// TwinCAT 3 PLC project GRAB
// ProgramVersion: 3.1.4024.12
// libraries:
//   CmpBitmapPool, * (System)
//   Tc2_MC2, * (Beckhoff Automation GmbH)
//   Tc2_Standard, * (Beckhoff Automation GmbH)
//   Tc2_System, * (Beckhoff Automation GmbH)
//   Tc3_Module, * (Beckhoff Automation GmbH)
//   VisuSymbols,3.5.10.0,System
// project tree:
//   / GlobalTextList.TcGTLO, ImagePool.TcIPO (not stored), PlcTask.TcTTO, Visualization Manager.TcVMO (not stored)
//   GVLs/ GVL.TcGVL, HAVL.TcGVL, RAVL.TcGVL, VAVL.TcGVL
//   POUs/ Homing.TcPOU, HorAxisPosCon.TcPOU, MAIN.TcPOU, ManualHorAxis.TcPOU, ManualRotAxis.TcPOU, ManualVerAxis.TcPOU, PositionHorAxis.TcPOU, PositionRotAxis.TcPOU, PositionVerAxis.TcPOU, POU.TcPOU, RunGRAB.TcPOU, Stop.TcPOU
//   VISUs/ Visualization.TcVIS
// real-time tasks:
//   TASK PlcTask: cycle T#10ms, priority 20, ADS port 350
// motion (NC):
//   TASK NC-Task 1 SAF: cycle T#2ms, priority 4, ADS port 501
//   TASK NC-Task 1 SVB: cycle T#10ms, priority 8, ADS port 511
//   AXIS HorizontalAxis (id 3)
//     Dynamic: AccelerationMaximum=2000, DecelerationMaximum=2000, Acceleration=100, Deceleration=500, Jerk=5000
//     Velo: RefSearch=80, RefSync=20, SlowManual=150, FastManual=150, Maximum=200
//     OtherSettings: AllowMotionCmdToSlave=true
//     encoder EncType=19
//       EncPara: ScaleFactorNumerator=0.004208, MaxCount=#xffffffff
//         SoftEndMinControl: Enable=true, Range=-100
//         SoftEndMaxControl: Enable=true, Range=700
//         Inc: RefSearchInverse=true, RefSyncInverse=false, RefSoftSyncMask=#x00000fff
//     drive DrvType=16
//       DrvPara: MaxCount=#xffffffff, DriveControlDWord=#x00020000
//         Analog: VeloReferenz=150, TorqueSetpointScale=10, ScaleFactorActTorque=0.1
//         TimeComp: TaskDelayCycles=1
//     controller CtrType=1
//       CtrPara: PriorControlFactor=1
//         PosDiffControl: Range=10
//         Observer: BandWidth=20
//   AXIS RotationAxis (id 4)
//     General: UnitName=Degree
//     Dynamic: AccelerationMaximum=20, DecelerationMaximum=20, Acceleration=10, Deceleration=50, Jerk=50
//     Velo: RefSearch=10, RefSync=5, SlowManual=20, FastManual=20, Maximum=21
//     OtherSettings: AllowMotionCmdToSlave=true, PulseDistancePos=0.05, PulseDistanceNeg=0.05
//     encoder EncType=19
//       EncPara: ScaleFactorNumerator=0.00505371, MaxCount=#xffffffff
//         SoftEndMinControl: Enable=true, Range=-100
//         SoftEndMaxControl: Enable=true, Range=100
//         Inc: RefSoftSyncMask=#x00000fff
//     drive DrvType=16
//       DrvPara: MaxCount=#xffffffff, DriveControlDWord=#x00020000
//         Analog: VeloReferenz=20, TorqueSetpointScale=10, ScaleFactorActTorque=0.1
//         TimeComp: TaskDelayCycles=1
//     controller CtrType=1
//       CtrPara: PriorControlFactor=1
//         Observer: BandWidth=20
//   AXIS VerticalAxis (id 5)
//     Dynamic: AccelerationMaximum=50, DecelerationMaximum=50, Acceleration=80, Deceleration=120, Jerk=6000
//     Velo: RefSearch=50, RefSync=10, SlowManual=150, FastManual=150, Maximum=200
//     OtherSettings: AllowMotionCmdToSlave=true
//     encoder EncType=19
//       EncPara: ScaleFactorNumerator=0.004208, Inverse=true, MaxCount=#xffffffff
//         SoftEndMinControl: Enable=true, Range=-50
//         SoftEndMaxControl: Enable=true, Range=1200
//         Inc: RefSearchInverse=true, RefSyncInverse=false, RefSoftSyncMask=#x00000fff
//     drive DrvType=16
//       DrvPara: Inverse=true, MaxCount=#xffffffff, DriveControlDWord=#x00020000
//         Analog: VeloReferenz=150, TorqueSetpointScale=10, ScaleFactorActTorque=0.1
//         TimeComp: TaskDelayCycles=1
//     controller CtrType=1
//       CtrPara: PriorControlFactor=1
//         PosDiffControl: Time=0.05
//         Observer: BandWidth=20
// I/O:
//   DEVICE Device 1 (EtherCAT), AmsNetId 5.46.12.154.2.1
//     Term 1 (EK1200) [EK1200-5000 EtherCAT Power supply (2A E-Bus)]
//       Term 2 (EL1008) [EL1008 8Ch. Dig. Input 24V, 3ms]
//       Term 3 (EL2008) [EL2008 8Ch. Dig. Output 24V, 0.5A]
//       Term 4 (EL1904) [EL1904, 4 Ch. Safety Input 24V, TwinSAFE]
//         modules: Module 1 (FSOES)
//       Term 5 (EK1110) [EK1110 EtherCAT extension]
//     Drive Hor (N5-2-1) [N5 EtherCAT Drive (CoE)]
//     Drive Rot (N5-2-1) [N5 EtherCAT Drive (CoE)]
//     Drive Ver (N5-2-1) [N5 EtherCAT Drive (CoE)]
// variable links:
//   NC-Task 1 SAF/Axes/HorizontalAxis <-> Device 1 (EtherCAT)/Drive Hor (N5-2-1)
//     Drive/Inputs/In/nState1 <-> Transmit PDO 1 Mapping Parameter/Statusword
//     Drive/Inputs/In/nState2 <-> Transmit PDO 1 Mapping Parameter/Statusword @bit 8
//     Drive/Inputs/In/nState4 @bit 1 <-> WcState/InputToggle
//     Drive/Inputs/In/nState4 <-> WcState/WcState
//     Drive/Inputs/In/nState5 <-> Transmit PDO 1 Mapping Parameter/Modes of operation display
//     Drive/Outputs/Out/nCtrl1 <-> Receive PDO 1 Mapping Parameter/Controlword
//     Drive/Outputs/Out/nCtrl2 <-> Receive PDO 1 Mapping Parameter/Controlword @bit 8
//     Drive/Outputs/Out/nCtrl5 <-> Receive PDO 1 Mapping Parameter/Modes of operation
//     Drive/Outputs/Out/nDataOut1 <-> Receive PDO 1 Mapping Parameter/Target Position
//     Enc/Inputs/In/nDataIn1 <-> Transmit PDO 1 Mapping Parameter/Position actual value
//     Enc/Inputs/In/nState4 @bit 1 <-> WcState/InputToggle
//     Enc/Inputs/In/nState4 <-> WcState/WcState
//   NC-Task 1 SAF/Axes/RotationAxis <-> Device 1 (EtherCAT)/Drive Rot (N5-2-1)
//     Drive/Inputs/In/nState1 <-> Transmit PDO 1 Mapping Parameter/Statusword
//     Drive/Inputs/In/nState2 <-> Transmit PDO 1 Mapping Parameter/Statusword @bit 8
//     Drive/Inputs/In/nState4 @bit 1 <-> WcState/InputToggle
//     Drive/Inputs/In/nState4 <-> WcState/WcState
//     Drive/Inputs/In/nState5 <-> Transmit PDO 1 Mapping Parameter/Modes of operation display
//     Drive/Outputs/Out/nCtrl1 <-> Receive PDO 1 Mapping Parameter/Controlword
//     Drive/Outputs/Out/nCtrl2 <-> Receive PDO 1 Mapping Parameter/Controlword @bit 8
//     Drive/Outputs/Out/nCtrl5 <-> Receive PDO 1 Mapping Parameter/Modes of operation
//     Drive/Outputs/Out/nDataOut1 <-> Receive PDO 1 Mapping Parameter/Target Position
//     Enc/Inputs/In/nDataIn1 <-> Transmit PDO 1 Mapping Parameter/Position actual value
//     Enc/Inputs/In/nState4 @bit 1 <-> WcState/InputToggle
//     Enc/Inputs/In/nState4 <-> WcState/WcState
//   NC-Task 1 SAF/Axes/VerticalAxis <-> Device 1 (EtherCAT)/Drive Ver (N5-2-1)
//     Drive/Inputs/In/nState1 <-> Transmit PDO 1 Mapping Parameter/Statusword
//     Drive/Inputs/In/nState2 <-> Transmit PDO 1 Mapping Parameter/Statusword @bit 8
//     Drive/Inputs/In/nState4 @bit 1 <-> WcState/InputToggle
//     Drive/Inputs/In/nState4 <-> WcState/WcState
//     Drive/Inputs/In/nState5 <-> Transmit PDO 1 Mapping Parameter/Modes of operation display
//     Drive/Outputs/Out/nCtrl1 <-> Receive PDO 1 Mapping Parameter/Controlword
//     Drive/Outputs/Out/nCtrl2 <-> Receive PDO 1 Mapping Parameter/Controlword @bit 8
//     Drive/Outputs/Out/nCtrl5 <-> Receive PDO 1 Mapping Parameter/Modes of operation
//     Drive/Outputs/Out/nDataOut1 <-> Receive PDO 1 Mapping Parameter/Target Position
//     Enc/Inputs/In/nDataIn1 <-> Transmit PDO 1 Mapping Parameter/Position actual value
//     Enc/Inputs/In/nState4 @bit 1 <-> WcState/InputToggle
//     Enc/Inputs/In/nState4 <-> WcState/WcState
//   GRAB/GRAB Instance <-> Device 1 (EtherCAT)/Drive Hor (N5-2-1)
//     PlcTask Outputs/HAVL.motorDriveSubmodeSelect <-> Receive PDO 1 Mapping Parameter/Motor drive submode select
//   GRAB/GRAB Instance <-> Device 1 (EtherCAT)/Drive Rot (N5-2-1)
//     PlcTask Outputs/RAVL.motorDriveSubmodeSelect <-> Receive PDO 1 Mapping Parameter/Motor drive submode select
//   GRAB/GRAB Instance <-> Device 1 (EtherCAT)/Drive Ver (N5-2-1)
//     PlcTask Outputs/VAVL.motorDriveSubmodeSelect <-> Receive PDO 1 Mapping Parameter/Motor drive submode select
//   GRAB/GRAB Instance <-> Device 1 (EtherCAT)/Term 1 (EK1200)/Term 2 (EL1008)
//     PlcTask Inputs/HAVL.endStop <-> Channel 1/Input
//     PlcTask Inputs/RAVL.endStop <-> Channel 3/Input
//     PlcTask Inputs/VAVL.endStopBottom <-> Channel 2/Input
//     PlcTask Inputs/VAVL.endStopTop <-> Channel 4/Input
//   GRAB/GRAB Instance <-> NC-Task 1 SAF/Axes/HorizontalAxis
//     PlcTask Inputs/HAVL.axis.NcToPlc <-> Outputs/ToPlc
//     PlcTask Outputs/HAVL.axis.PlcToNc <-> Inputs/FromPlc
//   GRAB/GRAB Instance <-> NC-Task 1 SAF/Axes/RotationAxis
//     PlcTask Inputs/RAVL.axis.NcToPlc <-> Outputs/ToPlc
//     PlcTask Outputs/RAVL.axis.PlcToNc <-> Inputs/FromPlc
//   GRAB/GRAB Instance <-> NC-Task 1 SAF/Axes/VerticalAxis
//     PlcTask Inputs/VAVL.axis.NcToPlc <-> Outputs/ToPlc
//     PlcTask Outputs/VAVL.axis.PlcToNc <-> Inputs/FromPlc

CONFIGURATION GRAB
    RESOURCE PLC ON TwinCAT3
        TASK PlcTask(INTERVAL := T#10ms, PRIORITY := 20);
        PROGRAM MAIN WITH PlcTask : MAIN;
    END_RESOURCE
END_CONFIGURATION

// ---- GVLs/GVL.TcGVL
{attribute 'qualified_only'}
VAR_GLOBAL
	stateGRAB: INT := 0;
	newStateGRAB: INT := 0;
	currentStateGRAB: INT;
	
	homingState: INT := 1;
	homingDone: BOOL := FALSE;
	
	stop: BOOL := FALSE;
END_VAR

// ---- GVLs/HAVL.TcGVL
{attribute 'qualified_only'}
VAR_GLOBAL
	axis: AXIS_REF;
	axisPower: MC_Power;
	axisMoveAbsolute: MC_MoveAbsolute;
	axisErrorReset: MC_Reset;
	axisReadActualPosition: MC_ReadActualPosition;
	axisMoveManual: MC_Jog;
	axisHome: MC_Home;
	axisStop: MC_Stop;
	
	enable: BOOL := FALSE;
	override: LREAL := 100;
	enableMove: BOOL := FALSE;
	targetPosition: LREAL := 0;
	targetVelocity: LREAL := 150;
	actualPosition: LREAL;
	actualPositionInt: INT;
	motorDriveSubmodeSelect AT%Q*:UDINT := 65;
	
	execute: BOOL := FALSE;
	extend: BOOL := FALSE;
	retract: BOOL := FALSE;
	busy: BOOL := FALSE;
	running: BOOL := FALSE;
	done: BOOL := FALSE;
	resetError: BOOL := FALSE;
	currentError: UDINT;
	currentErrorPower: UDINT;
	currentErrorCommand: UDINT;
	stopped: BOOL := FALSE;
	
	lastExtend: BOOL := FALSE;
	lastRetract: BOOL := FALSE;
	
	endStop AT %I*: BOOL;
	
	homePosition: LREAL := 0;
END_VAR

// ---- GVLs/RAVL.TcGVL
{attribute 'qualified_only'}
VAR_GLOBAL
	axis: AXIS_REF;
	axisPower: MC_Power;
	axisMoveAbsolute: MC_MoveAbsolute;
	axisErrorReset: MC_Reset;
	axisReadActualPosition: MC_ReadActualPosition;
	axisMoveManual: MC_Jog;
	axisHome: MC_Home;
	axisStop: MC_Stop;
	
	enable: BOOL := FALSE;
	override: LREAL := 100;
	enableMove: BOOL := FALSE;
	targetPosition: LREAL := 0;
	targetVelocity: LREAL := 20;
	actualPosition: LREAL;
	actualPositionInt: INT;
	motorDriveSubmodeSelect AT%Q*:UDINT := 65;
	
	execute: BOOL := FALSE;
	clockwise: BOOL := FALSE;
	counterClockwise: BOOL := FALSE;
	busy: BOOL := FALSE;
	running: BOOL := FALSE;
	done: BOOL := FALSE;
	resetError: BOOL := FALSE;
	currentError: UDINT;
	currentErrorPower: UDINT;
	currentErrorCommand: UDINT;
	stopped: BOOL := FALSE;
	
	lastClockwise: BOOL := FALSE;
	lastCounterClockwise: BOOL := FALSE;
	
	endStop AT %I*: BOOL;
	
	homePosition: LREAL := 80;
END_VAR

// ---- GVLs/VAVL.TcGVL
{attribute 'qualified_only'}
VAR_GLOBAL
	axis: AXIS_REF;
	axisPower: MC_Power;
	axisMoveAbsolute: MC_MoveAbsolute;
	axisErrorReset: MC_Reset;
	axisReadActualPosition: MC_ReadActualPosition;
	axisMoveManual: MC_Jog;
	axisHome: MC_Home;
	axisStop: MC_Stop;
	
	enable: BOOL := FALSE;
	override: LREAL := 100;
	enableMove: BOOL := FALSE;
	targetPosition: LREAL := 0;
	targetVelocity: LREAL := 200;
	actualPosition: LREAL;
	actualPositionInt: INT;
	motorDriveSubmodeSelect AT%Q*:UDINT := 68;
	
	execute: BOOL := FALSE;
	ascend: BOOL := FALSE;
	descend: BOOL := FALSE;
	busy: BOOL := FALSE;
	running: BOOL := FALSE;
	done: BOOL := FALSE;
	resetError: BOOL := FALSE;
	currentError: UDINT;
	currentErrorPower: UDINT;
	currentErrorCommand: UDINT;
	stopped: BOOL := FALSE;
	
	homePosition: LREAL := 0;	

	endStopTop AT %I*: BOOL;
	endStopBottom AT %I*: BOOL;
	brake AT %Q*: BOOL;
END_VAR

// ---- POUs/MAIN.TcPOU
PROGRAM MAIN
VAR
END_VAR

RunGRAB();

END_PROGRAM

// ---- POUs/RunGRAB.TcPOU
PROGRAM RunGRAB
VAR

END_VAR
VAR CONSTANT 
    HOMING: INT := 1;
	MANUAL: INT := 2;
	POSITION: INT := 3;
END_VAR

IF(HAVL.stopped OR RAVL.stopped OR VAVL.stopped) THEN
	GVL.stateGRAB := 0;
END_IF

// State machine
CASE GVL.stateGRAB OF
HOMING:
	.Homing();
	
MANUAL:
	.ManualHorAxis();
	.ManualRotAxis();
	.ManualVerAxis();
	
POSITION:
	.PositionHorAxis();
	.PositionRotAxis();
	.PositionVerAxis();

ELSE
	// GRAB waiting for command
END_CASE

HAVL.axisStop(
	Axis:=HAVL.axis,
	Execute:=GVL.stop,
	Deceleration:=100,
	Jerk:=5000,
	Options:=,
	Done=>,
	Busy=>HAVL.stopped,
	Active=>,
	CommandAborted=>,
	Error=>,
	ErrorID=>
	);
	
RAVL.axisStop(
	Axis:=RAVL.axis,
	Execute:=GVL.stop,
	Deceleration:=100,
	Jerk:=5000,
	Options:=,
	Done=>,
	Busy=>RAVL.stopped,
	Active=>,
	CommandAborted=>,
	Error=>,
	ErrorID=>
	);
	
VAVL.axisStop(
	Axis:=VAVL.axis,
	Execute:=GVL.stop,
	Deceleration:=100,
	Jerk:=5000,
	Options:=,
	Done=>,
	Busy=>VAVL.stopped,
	Active=>,
	CommandAborted=>,
	Error=>,
	ErrorID=>
	);

END_PROGRAM

// ---- POUs/Homing.TcPOU
PROGRAM Homing
VAR
	horAxisHomingDone: BOOL := FALSE;
	rotAxisHomingDone: BOOL := FALSE;
	verAxisHomingDone: BOOL := FALSE;
	lastTime: TIME;
	timerOn: BOOL := FALSE;
END_VAR
VAR CONSTANT 
    HOME_SNAKE: INT := 1;
	HOME_SNAKEBOX: INT := 2;
	HOME_VERTICAL: INT := 3;
END_VAR

// State machine
HAVL.axis.ReadStatus();
RAVL.axis.ReadStatus();
VAVL.axis.ReadStatus();
CASE GVL.homingState OF
HOME_SNAKE:
	timerOn:= FALSE;
	IF horAxisHomingDone THEN
		HAVL.enable := FALSE;
		GVL.homingState := 2;
	ELSE
		HAVL.enable := TRUE;
	END_IF
	
	HAVL.axisPower(
		Axis:= HAVL.axis,
		Enable:= HAVL.enable,
		Enable_Positive:= HAVL.enable,
		Enable_Negative:= HAVL.enable,
		Override:= HAVL.override,
		BufferMode:= ,
		Options:= ,
		Status=> HAVL.running,
		Busy=> ,
		Active=> ,
		Error=> ,
		ErrorID=> HAVL.currentErrorPower
	);
	
	HAVL.axisHome(
		Axis:= HAVL.axis,
		Execute:= HAVL.execute,
		Position:= HAVL.homePosition,
		HomingMode:= MC_DefaultHoming,
		BufferMode:= ,
		Options:= ,
		bCalibrationCam:= HAVL.endStop,
		Done=> HAVL.done,
		Busy=> HAVL.busy,
		Active=> ,
		CommandAborted=> ,
		Error=> ,
		ErrorID=> HAVL.currentErrorCommand
	);
	
	IF HAVL.running AND NOT(HAVL.busy) AND NOT(horAxisHomingDone) THEN
		HAVL.execute := TRUE;
	ELSE
		HAVL.execute := FALSE;
	END_IF
	
	IF HAVL.done THEN
		horAxisHomingDone := TRUE;
		RAVL.enable := TRUE;
	END_IF
		
HOME_SNAKEBOX:
	// do some invers motor shit	
	horAxisHomingDone := FALSE;
	
	IF rotAxisHomingDone THEN
		RAVL.enable := FALSE;
		GVL.homingState := 3;
	ELSE
		RAVL.enable := TRUE;
	END_IF
	
	RAVL.axisPower(
		Axis:= RAVL.axis,
		Enable:= RAVL.enable,
		Enable_Positive:= RAVL.enable,
		Enable_Negative:= RAVL.enable,
		Override:= RAVL.override,
		BufferMode:= ,
		Options:= ,
		Status=> RAVL.running,
		Busy=> ,
		Active=> ,
		Error=> ,
		ErrorID=> RAVL.currentErrorPower
	);
	
	RAVL.axisHome(
		Axis:= RAVL.axis,
		Execute:= RAVL.execute,
		Position:= RAVL.homePosition,
		HomingMode:= MC_DefaultHoming,
		BufferMode:= ,
		Options:= ,
		bCalibrationCam:= RAVL.endStop,
		Done=> RAVL.done,
		Busy=> RAVL.busy,
		Active=> ,
		CommandAborted=> ,
		Error=> ,
		ErrorID=> RAVL.currentErrorCommand
	);
	
	IF RAVL.running AND NOT(RAVL.busy) AND NOT(rotAxisHomingDone) THEN
		RAVL.execute := TRUE;
	ELSE
		RAVL.execute := FALSE;
	END_IF
	
	IF RAVL.done THEN
		rotAxisHomingDone := TRUE;
		//VAVL.enable := TRUE;
	END_IF
	
HOME_VERTICAL:
	//SAMELUR
	rotAxisHomingDone := FALSE;
	
	IF verAxisHomingDone THEN
		VAVL.enable := FALSE;
		GVL.homingState := 1;
		GVL.stateGRAB := 0;
		GVL.homingDone := TRUE;
		verAxisHomingDone := FALSE;
	ELSE
		VAVL.enable := TRUE;
	END_IF
	
	VAVL.axisPower(
		Axis:= VAVL.axis,
		Enable:= VAVL.enable,
		Enable_Positive:= VAVL.enable,
		Enable_Negative:= VAVL.enable,
		Override:= VAVL.override,
		BufferMode:= ,
		Options:= ,
		Status=> VAVL.running,
		Busy=> ,
		Active=> ,
		Error=> ,
		ErrorID=> VAVL.currentErrorPower
	);
	
	VAVL.axisHome(
		Axis:= VAVL.axis,
		Execute:= VAVL.execute,
		Position:= VAVL.homePosition,
		HomingMode:= MC_DefaultHoming,
		BufferMode:= ,
		Options:= ,
		bCalibrationCam:= NOT(VAVL.endStopBottom),
		Done=> VAVL.done,
		Busy=> VAVL.busy,
		Active=> ,
		CommandAborted=> ,
		Error=> ,
		ErrorID=> VAVL.currentErrorCommand
	);
	
	IF VAVL.running AND NOT(timerOn) AND NOT(VAVL.busy) AND NOT(verAxisHomingDone) THEN
		lastTime := TIME() + T#3S;
		timerOn := TRUE;
	END_IF
	
	IF VAVL.running AND NOT(VAVL.busy) AND NOT(verAxisHomingDone) AND (TIME()>lastTime) AND timerOn THEN
		VAVL.execute := TRUE;
		timerOn := FALSE;
	ELSE
		VAVL.execute := FALSE;
	END_IF
	
	IF VAVL.done THEN
		verAxisHomingDone := TRUE;
	END_IF

ELSE
	// GRAB waiting for command
END_CASE

END_PROGRAM

// ---- POUs/ManualHorAxis.TcPOU
PROGRAM ManualHorAxis
VAR
END_VAR

HAVL.axis.ReadStatus();

IF HAVL.extend AND NOT(HAVL.endStop) THEN
	HAVL.lastExtend := TRUE;
	HAVL.lastRetract := FALSE;
END_IF

IF HAVL.retract AND NOT(HAVL.endStop) THEN
	HAVL.lastExtend := FALSE;
	HAVL.lastRetract := TRUE;
END_IF

HAVL.axisPower(
	Axis:= HAVL.axis,
	Enable:= HAVL.enable,
	Enable_Positive:= HAVL.enable,
	Enable_Negative:= HAVL.enable,
	Override:= HAVL.override,
	BufferMode:= ,
	Options:= ,
	Status=> HAVL.running,
	Busy=> ,
	Active=> ,
	Error=> ,
	ErrorID=> HAVL.currentErrorPower
);

HAVL.axisMoveManual(
	Axis:= HAVL.axis,
	JogForward:= (HAVL.extend AND (NOT(HAVL.endStop) OR (HAVL.endStop AND HAVL.lastRetract))),
	JogBackwards:= (HAVL.retract AND (NOT(HAVL.endStop) OR (HAVL.endStop AND HAVL.lastExtend))),
	Mode:= ,
	Position:= ,
	Velocity:= ,
	Acceleration:= ,
	Deceleration:= ,
	Jerk:= ,
	Done=> HAVL.done,
	Busy=> HAVL.busy,
	Active=> ,
	CommandAborted=> ,
	Error=> ,
	ErrorID=> HAVL.currentErrorCommand
);
	
IF HAVL.busy THEN
	HAVL.axisReadActualPosition(Axis := HAVL.axis, Enable := TRUE, Valid=>, Busy=>, Error=>, ErrorID=>, Position=> HAVL.actualPosition);
END_IF
HAVL.actualPositionInt := LREAL_TO_INT(HAVL.actualPosition);

HAVL.axisErrorReset(Axis := HAVL.axis, Execute := HAVL.resetError, Done =>, Error =>, ErrorID => HAVL.currentError);

END_PROGRAM

// ---- POUs/ManualRotAxis.TcPOU
PROGRAM ManualRotAxis
VAR
END_VAR

RAVL.axis.ReadStatus();

IF RAVL.clockwise AND NOT(RAVL.endStop) THEN
	RAVL.lastClockwise := TRUE;
	RAVL.lastCounterClockwise := FALSE;
END_IF

IF RAVL.counterClockwise AND NOT(RAVL.endStop) THEN
	RAVL.lastClockwise := FALSE;
	RAVL.lastCounterClockwise := TRUE;
END_IF

RAVL.axisPower(
	Axis:= RAVL.axis,
	Enable:= RAVL.enable,
	Enable_Positive:= RAVL.enable,
	Enable_Negative:= RAVL.enable,
	Override:= RAVL.override,
	BufferMode:= ,
	Options:= ,
	Status=> RAVL.running,
	Busy=> ,
	Active=> ,
	Error=> ,
	ErrorID=> RAVL.currentErrorPower
);

RAVL.axisMoveManual(
	Axis:= RAVL.axis,
	JogForward:= (RAVL.counterClockwise AND (NOT(RAVL.endStop) OR (RAVL.endStop AND RAVL.lastClockwise))),
	JogBackwards:= (RAVL.clockwise AND (NOT(RAVL.endStop) OR (RAVL.endStop AND RAVL.lastCounterClockwise))),
	Mode:= ,
	Position:= ,
	Velocity:= ,
	Acceleration:= ,
	Deceleration:= ,
	Jerk:= ,
	Done=> RAVL.done,
	Busy=> RAVL.busy,
	Active=> ,
	CommandAborted=> ,
	Error=> ,
	ErrorID=> RAVL.currentErrorCommand
);

IF RAVL.busy THEN
	RAVL.axisReadActualPosition(Axis := RAVL.axis, Enable := TRUE, Valid=>, Busy=>, Error=>, ErrorID=>, Position=> RAVL.actualPosition);
END_IF
RAVL.actualPositionInt := LREAL_TO_INT(RAVL.actualPosition);

RAVL.axisErrorReset(Axis := RAVL.axis, Execute := RAVL.resetError, Done =>, Error =>, ErrorID => RAVL.currentError);

END_PROGRAM

// ---- POUs/ManualVerAxis.TcPOU
PROGRAM ManualVerAxis
VAR
END_VAR

VAVL.axis.ReadStatus();


VAVL.axisPower(
	Axis:= VAVL.axis,
	Enable:= VAVL.enable,
	Enable_Positive:= VAVL.enable,
	Enable_Negative:= VAVL.enable,
	Override:= VAVL.override,
	BufferMode:= ,
	Options:= ,
	Status=> VAVL.running,
	Busy=> ,
	Active=> ,
	Error=> ,
	ErrorID=> VAVL.currentErrorPower
);

VAVL.axisMoveManual(
	Axis:= VAVL.axis,
	JogForward:= (VAVL.ascend AND VAVL.endStopTop),
	JogBackwards:= (VAVL.descend AND VAVL.endStopBottom),
	Mode:= ,
	Position:= ,
	Velocity:= ,
	Acceleration:= ,
	Deceleration:= ,
	Jerk:= ,
	Done=> VAVL.done,
	Busy=> VAVL.busy,
	Active=> ,
	CommandAborted=> ,
	Error=> ,
	ErrorID=> VAVL.currentErrorCommand
);
	
IF VAVL.busy THEN
	VAVL.axisReadActualPosition(Axis := VAVL.axis, Enable := TRUE, Valid=>, Busy=>, Error=>, ErrorID=>, Position=> VAVL.actualPosition);
END_IF
VAVL.actualPositionInt := LREAL_TO_INT(VAVL.actualPosition);

VAVL.axisErrorReset(Axis := VAVL.axis, Execute := VAVL.resetError, Done =>, Error =>, ErrorID => VAVL.currentError);

END_PROGRAM

// ---- POUs/PositionHorAxis.TcPOU
PROGRAM PositionHorAxis
VAR
END_VAR

HAVL.axis.ReadStatus();

HAVL.axisPower(
	Axis:= HAVL.axis,
	Enable:= HAVL.enable,
	Enable_Positive:= HAVL.enable,
	Enable_Negative:= HAVL.enable,
	Override:= HAVL.override,
	BufferMode:= ,
	Options:= ,
	Status=> HAVL.running,
	Busy=> ,
	Active=> ,
	Error=> ,
	ErrorID=> HAVL.currentErrorPower
);

HAVL.axisMoveAbsolute(
	Axis:= HAVL.axis,
	Execute:= HAVL.enableMove,
	Position:= HAVL.targetPosition,
	Velocity:= HAVL.targetVelocity,
	Acceleration:= ,
	Deceleration:= ,
	Jerk:= ,
	BufferMode:= ,
	Options:= ,
	Done=> HAVL.done,
	Busy=> HAVL.busy,
	Active=> ,
	CommandAborted=> ,
	Error=> ,
	ErrorID=> HAVL.currentErrorCommand 
);

IF HAVL.busy THEN
	HAVL.axisReadActualPosition(Axis := HAVL.axis, Enable := TRUE, Valid=>, Busy=>, Error=>, ErrorID=>, Position=> HAVL.actualPosition);
END_IF
HAVL.actualPositionInt := LREAL_TO_INT(HAVL.actualPosition);

HAVL.axisErrorReset(Axis := HAVL.axis, Execute := HAVL.resetError, Done =>, Error =>, ErrorID => HAVL.currentError);

END_PROGRAM

// ---- POUs/PositionRotAxis.TcPOU
PROGRAM PositionRotAxis
VAR
END_VAR

RAVL.axis.ReadStatus();

RAVL.axisPower(
	Axis:= RAVL.axis,
	Enable:= RAVL.enable,
	Enable_Positive:= RAVL.enable,
	Enable_Negative:= RAVL.enable,
	Override:= RAVL.override,
	BufferMode:= ,
	Options:= ,
	Status=> RAVL.running,
	Busy=> ,
	Active=> ,
	Error=> ,
	ErrorID=> RAVL.currentErrorPower
);

RAVL.axisMoveAbsolute(
	Axis:= RAVL.axis,
	Execute:= RAVL.enableMove,
	Position:= RAVL.targetPosition,
	Velocity:= RAVL.targetVelocity,
	Acceleration:= ,
	Deceleration:= ,
	Jerk:= ,
	BufferMode:= ,
	Options:= ,
	Done=> RAVL.done,
	Busy=> RAVL.busy,
	Active=> ,
	CommandAborted=> ,
	Error=> ,
	ErrorID=> RAVL.currentErrorCommand 
);

IF RAVL.busy THEN
	RAVL.axisReadActualPosition(Axis := RAVL.axis, Enable := TRUE, Valid=>, Busy=>, Error=>, ErrorID=>, Position=> RAVL.actualPosition);
END_IF
RAVL.actualPositionInt := LREAL_TO_INT(RAVL.actualPosition);

RAVL.axisErrorReset(Axis := RAVL.axis, Execute := RAVL.resetError, Done =>, Error =>, ErrorID => RAVL.currentError);

END_PROGRAM

// ---- POUs/PositionVerAxis.TcPOU
PROGRAM PositionVerAxis
VAR
END_VAR

VAVL.axis.ReadStatus();

VAVL.axisPower(
	Axis:= VAVL.axis,
	Enable:= VAVL.enable,
	Enable_Positive:= VAVL.enable,
	Enable_Negative:= VAVL.enable,
	Override:= VAVL.override,
	BufferMode:= ,
	Options:= ,
	Status=> VAVL.running,
	Busy=> ,
	Active=> ,
	Error=> ,
	ErrorID=> VAVL.currentErrorPower
);

VAVL.axisMoveAbsolute(
	Axis:= VAVL.axis,
	Execute:= VAVL.enableMove,
	Position:= VAVL.targetPosition,
	Velocity:= VAVL.targetVelocity,
	Acceleration:= ,
	Deceleration:= ,
	Jerk:= ,
	BufferMode:= ,
	Options:= ,
	Done=> VAVL.done,
	Busy=> VAVL.busy,
	Active=> ,
	CommandAborted=> ,
	Error=> ,
	ErrorID=> VAVL.currentErrorCommand 
);

IF VAVL.busy THEN
	VAVL.axisReadActualPosition(Axis := VAVL.axis, Enable := TRUE, Valid=>, Busy=>, Error=>, ErrorID=>, Position=> VAVL.actualPosition);
END_IF
VAVL.actualPositionInt := LREAL_TO_INT(VAVL.actualPosition);

VAVL.axisErrorReset(Axis := VAVL.axis, Execute := VAVL.resetError, Done =>, Error =>, ErrorID => VAVL.currentError);

END_PROGRAM

// ---- POUs/Stop.TcPOU
PROGRAM Stop
VAR
END_VAR
VAR CONSTANT 
    STOP_ALL_AXIS: INT := 1;
	RESET_STOP: INT := 2;
END_VAR

HAVL.axis.ReadStatus();
RAVL.axis.ReadStatus();
VAVL.axis.ReadStatus();

HAVL.axisStop(
	Axis:=HAVL.axis,
	Execute:=HAVL.execute,
	Deceleration:=100,
	Jerk:=5000,
	Options:=,
	Done=>,
	Busy=>,
	Active=>,
	CommandAborted=>,
	Error=>,
	ErrorID=>
	);
	
RAVL.axisStop(
	Axis:=RAVL.axis,
	Execute:=RAVL.execute,
	Deceleration:=100,
	Jerk:=5000,
	Options:=,
	Done=>,
	Busy=>,
	Active=>,
	CommandAborted=>,
	Error=>,
	ErrorID=>
	);
	
VAVL.axisStop(
	Axis:=VAVL.axis,
	Execute:=VAVL.execute,
	Deceleration:=100,
	Jerk:=5000,
	Options:=,
	Done=>,
	Busy=>,
	Active=>,
	CommandAborted=>,
	Error=>,
	ErrorID=>
	);

END_PROGRAM

// ---- POUs/HorAxisPosCon.TcPOU
PROGRAM HorAxisPosCon
VAR
	running: BOOL := FALSE;
	busy: BOOL := TRUE;
	done: bool := TRUE;
	
	fbTimer: TON;
	tTimerValue     : TIME := T#5S;
	bStart          : BOOL := TRUE;
	
	reset: BOOL := FALSE;
	
	currentError: UDINT;
	
	start: BOOL := FALSE;
	position: LREAL;
	count: INT := 0;
END_VAR

HAVL.axis.ReadStatus();

fbTimer(IN := bStart, PT := tTimerValue);
IF done THEN
	bStart := TRUE;
END_IF

IF start AND NOT(busy) THEN
	HAVL.enable := TRUE;
ELSIF NOT(start) AND NOT(busy) THEN
	HAVL.enable := FALSE;
END_IF

HAVL.axisPower(
	Axis:= HAVL.axis,
	Enable:= HAVL.enable,
	Enable_Positive:= HAVL.enable,
	Enable_Negative:= HAVL.enable,
	Override:= HAVL.override,
	BufferMode:= ,
	Options:= ,
	Status=> running,
	Busy=> ,
	Active=> ,
	Error=> ,
	ErrorID=> currentError
);

HAVL.axisMoveAbsolute(
	Axis:= HAVL.axis,
	Execute:= HAVL.enableMove,
	Position:= HAVL.targetPosition,
	Velocity:= HAVL.targetVelocity,
	Acceleration:= ,
	Deceleration:= ,
	Jerk:= ,
	BufferMode:= ,
	Options:= ,
	Done=> done,
	Busy=> busy,
	Active=> ,
	CommandAborted=> ,
	Error=> ,
	ErrorID=> currentError 
);

IF NOT(busy) AND NOT(HAVL.enableMove)AND running AND HAVL.enable AND fbTimer.Q THEN
	HAVL.enableMove := TRUE;
	bStart := FALSE;
	IF HAVL.targetPosition = 0 THEN
		HAVL.targetPosition := 100;
	ELSE
		HAVL.targetPosition := 0;
	END_IF
END_IF

IF busy AND HAVL.enableMove THEN
	HAVL.enableMove := FALSE;
END_IF

HAVL.axisErrorReset(Axis := HAVL.axis, Execute := reset, Done =>, Error =>, ErrorID => currentError);

HAVL.axisReadActualPosition(Axis := HAVL.axis, Enable := busy, Valid=>, Busy=>, Error=>, ErrorID=>, Position=> position);

END_PROGRAM

// ---- POUs/POU.TcPOU
PROGRAM POU
VAR
	running: BOOL;
	currentError: UDINT;
	done: BOOL;
	busy: BOOL;
	reset: BOOL;
	position: LREAL;
END_VAR

HAVL.axis.ReadStatus();

HAVL.axisPower(
	Axis:= HAVL.axis,
	Enable:= HAVL.enable,
	Enable_Positive:= HAVL.enable,
	Enable_Negative:= HAVL.enable,
	Override:= HAVL.override,
	BufferMode:= ,
	Options:= ,
	Status=> running,
	Busy=> ,
	Active=> ,
	Error=> ,
	ErrorID=> currentError
);

HAVL.axisMoveAbsolute(
	Axis:= HAVL.axis,
	Execute:= HAVL.enableMove,
	Position:= HAVL.targetPosition,
	Velocity:= HAVL.targetVelocity,
	Acceleration:= ,
	Deceleration:= ,
	Jerk:= ,
	BufferMode:= ,
	Options:= ,
	Done=> done,
	Busy=> busy,
	Active=> ,
	CommandAborted=> ,
	Error=> ,
	ErrorID=> currentError 
);

HAVL.axisErrorReset(Axis := HAVL.axis, Execute := reset, Done =>, Error =>, ErrorID => currentError);

HAVL.axisReadActualPosition(Axis := HAVL.axis, Enable := busy, Valid=>, Busy=>, Error=>, ErrorID=>, Position=> position);

END_PROGRAM

// ---- GlobalTextList.TcGTLO
TEXTLIST GlobalTextList
  369 = 'Blir brukt fer å skru på aksen!'
  167 = 'Fram'
  355 = 'Skru på na aksen fer faen!'
  238 = 'When u dont want PP'
  114 = 'When you dont want the PP'
  778 = 'Å so tebake igjen'
END_TEXTLIST

// ---- VISUs/Visualization.TcVIS
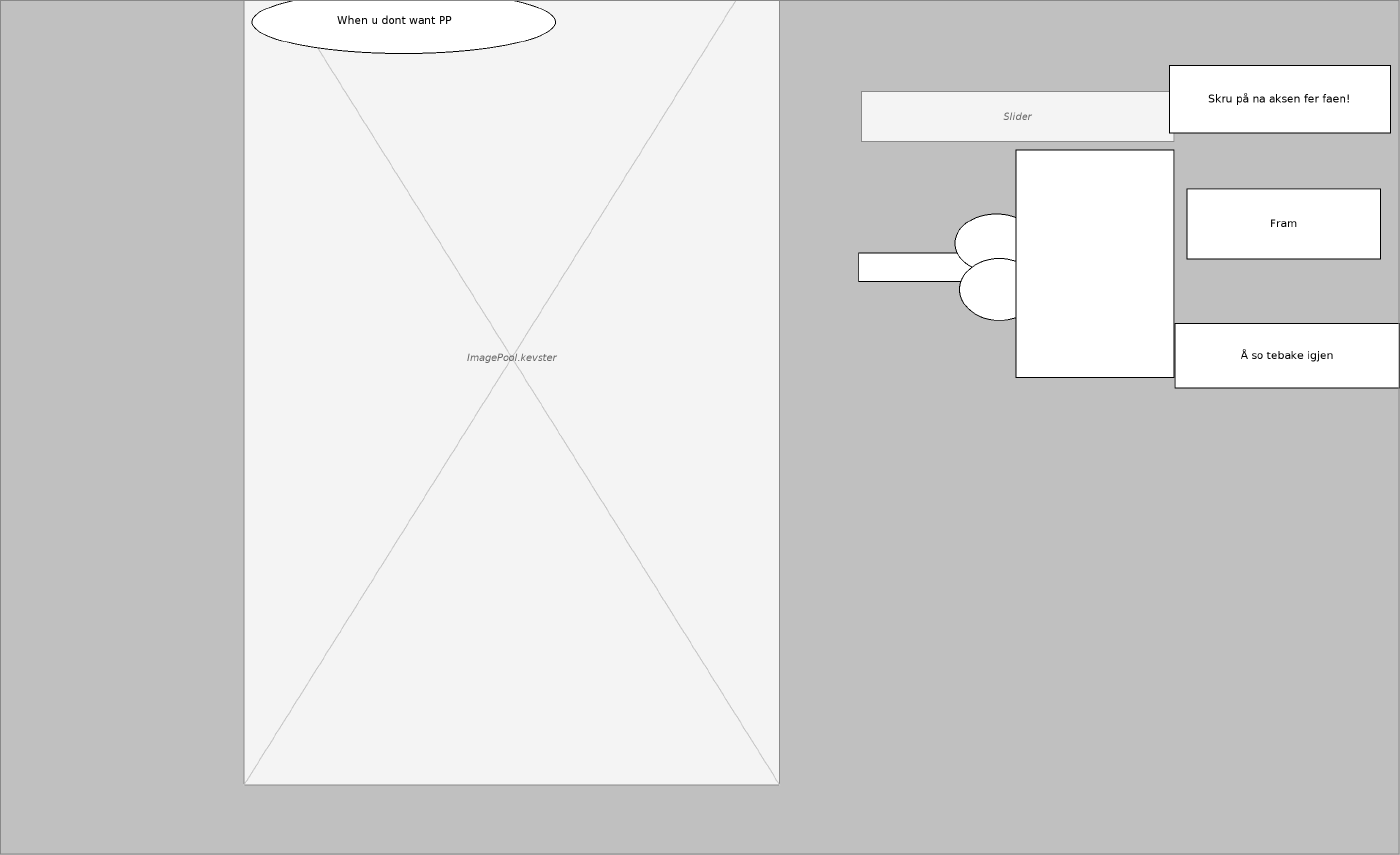
VISUALIZATION Visualization  // 1442x881
    Image (251,-72 552x881), image: ImagePool.kevster
    RoundedRectangle (884,260 312x30)
        p3528305787: -HAVL.actualPosition/10
    Ellipse (983,220 86x61)
    Ellipse (988,266 82x64)
    Slider (887,94 322x52), scale 0..100
    RoundedRectangle (1204,67 228x70), "Skru på na aksen fer faen!", tooltip "Blir brukt fer å skru på aksen!"
        toggle HAVL.enable
    RoundedRectangle (1222,194 200x73), "Fram"
        toggle HAVL.forward
    RoundedRectangle (1210,333 232x67), "Å so tebake igjen"
        toggle HAVL.retract
    Ellipse (259,-10 313x65)
    Label (331,6 150x30), "When u dont want PP"
    RoundedRectangle (1046,154 163x235)
END_VISUALIZATION
